FUNCTION_BLOCK Killer_Object EXTENDS Person_Object
VAR_INPUT
END_VAR
VAR_OUTPUT
END_VAR
VAR
    _isAlive : BOOL := TRUE;
    _Kill : Kill_Task(THIS^);
END_VAR

PROPERTY IsAlive : Bool
GET
IsAlive := _isAlive;
END_GET
SET
_isAlive := IsAlive;
END_SET
END_PROPERTY

METHOD Kill : TcoCore.ITcoTask
VAR_INPUT
    _Object2bKilled : REFERENCE TO Horse_Object;
END_VAR
_Kill(_Object2bKilled := _Object2bKilled, _Killer := THIS^);
Kill := _Kill;
END_METHOD

END_FUNCTION_BLOCK

(* stored: Version 1.1.0.1, ProductVersion 3.1.4024.9
   POU Killer_Object: Id {6cf1f058-fc3f-01f7-18ab-723f0f024201}, SpecialFunc None
   Property IsAlive: Id {8fc5e1d4-adfe-007f-142b-702cd6733a4d}
   Get Get: Id {4a59e1e1-9eb0-0bbd-09da-d20a1f70c7da}
   Set Set: Id {461e740a-66d2-00f6-2f6f-366a32c6bc80}
   Method Kill: Id {7893e1a3-6b2a-0373-30e3-e4bcb9cb5154} *)
